{attribute 'qualified_only'}
{attribute 'strict'}
TYPE E_General_ProcessCycle :
(
	
IDLE							,
CLOSE_PROCESS_DOOR				,
WAIT_CLOSE_PROCESS_DOOR			,
OPEN_PROCESS_DOOR				,
WAIT_OPEN_PROCESS_DOOR			,
EXTEND_PROCESS_CYLINDER			,
WAIT_EXTEND_PROCESS_CYLINDER	,
RETRACT_PROCESS_CYLINDER		,
WAIT_RETRACT_PROCESS_CYLINDER	,
RETRACT_MIDDLE_PROCESS_CYLINDER		,
WAIT_RETRACT_MIDDLE_PROCESS_CYLINDER	,
MOVE_NEST_TO_RIGHT				,
WAIT_MOVE_NEST_TO_RIGHT			,
MOVE_NEST_TO_LEFT				,
WAIT_MOVE_NEST_TO_LEFT			,
LEAK_TEST						,
WAIT_LEAK_TEST					,
HEIGHT_TEST						,
WAIT_HEIGHT_TEST				,
WAIT_TO_SAVE_DATA				,
WAIT_RESULTS					,
RESULTS							,
SAVE_DATA						,
SAVE_DATA2						,
CSV_NEST1						,
CSV_NEST2						,
WAIT_REJECT_PART				,

RESET_ALL_CMD						

);
END_TYPE

(* stored: Version 1.1.0.1, ProductVersion 3.1.4026.18
   DUT E_General_ProcessCycle: Id {efc1fb3f-e466-425d-af8e-a4df616b7389} *)
